PROGRAM MAIN
VAR
	fbi_lsm_main: fb_lsm_main;
	fbi_text_control_run: fb_text_control;
END_VAR

fbi_lsm_main();
fbi_text_control_run();

END_PROGRAM

(* stored: Version 1.1.0.1, ProductVersion 3.1.4024.12
   POU MAIN: Id {c726c6cb-38f1-459f-90ce-2fd1cbc12234}, SpecialFunc None *)
